// TIA Portal V17 export
// export: Created 2025-03-12T15:37:46.0301049Z, ExportSetting WithDefaults, DisplayName Totally Integrated Automation Portal, DisplayVersion V17 Update 8, DisplayName TIA Portal Openness, DisplayVersion V17 Update 8, DisplayName TIA Portal Version Control Interface, DisplayVersion V17, DisplayName SINAMICS Startdrive Advanced, DisplayVersion V17 SP2, DisplayName SINAMICS Startdrive G110M, G120, G120C, G120D, G120P, G115D, DisplayVersion V17 SP2, DisplayName SINAMICS Startdrive G130, G150, S120, S150, SINAMICS MV, S210, DisplayVersion V17 SP2, DisplayName STEP 7 Professional, DisplayVersion V17 Update 8, DisplayName SINUMERIK ONE STEP 7 Toolbox, DisplayVersion V17 Update 12, DisplayName SINUMERIK 840D sl STEP 7 Toolbox, DisplayVersion V17 Update 12, DisplayName STEP 7 Safety, DisplayVersion V17 Update 6, DisplayName WinCC Advanced, DisplayVersion V17 Update 8
TYPE "POWDER FEEDER HEATER JKT"
// stored: IsFailsafeCompliant false
   STRUCT
      START_GENERAL_CONDITIONS : Bool;   // Start General Conditions / START GENERAL CONDITIONS
      START_INITIAL_CONDITIONS_LINE_1 : Bool;   // Start Initial Conditions / START INITIAL CONDITIONS LINE 1
      START_INITIAL_CONDITIONS_LINE_2 : Bool;   // Start Initial Conditions / START INITIAL CONDITIONS LINE 2
      START_MANUAL_REQUEST_LINE_1 : Bool;   // Start Manual Request / START MANUAL REQUEST LINE 1
      START_MANUAL_REQUEST_LINE_2 : Bool;   // Start Manual Request / START MANUAL REQUEST LINE 2
      START_AUTO_REQUEST : Bool;   // Start Auto Request / START AUTO REQUEST
      START_GLOBAL_REQUEST_LINE_1 : Bool;   // Start Global Request / START GLOBAL REQUEST LINE 1
      START_GLOBAL_REQUEST_LINE_2 : Bool;   // Start Global Request / START GLOBAL REQUEST LINE 2
      START_COMMAND_LINE_1 : Bool;   // Start Command / START COMMAND LINE 1
      START_COMMAND_LINE_2 : Bool;   // Start Command / START COMMAND LINE 2
      START_LINE_1 : Bool;   // Start / START LINE 1
      START_LINE_2 : Bool;   // Start / START LINE 2
      FEEDBACK_ON_LINE_1 : Bool;   // Feedback On / FEEDBACK ON LINE 1
      FEEDBACK_ON_LINE_2 : Bool;   // Feedback On / FEEDBACK ON LINE 2
      STOP_GENERAL_CONDITIONS : Bool;   // Stop General Conditions / STOP GENERAL CONDITIONS
      STOP_INITIAL_CONDITIONS_LINE_1 : Bool;   // Stop Initial Conditions / STOP INITIAL CONDITIONS LINE 1
      STOP_INITIAL_CONDITIONS_LINE_2 : Bool;   // Stop Initial Conditions / STOP INITIAL CONDITIONS LINE 2
      STOP_MANUAL_REQUEST_LINE_1 : Bool;   // Stop Manual Request / STOP MANUAL REQUEST LINE 1
      STOP_MANUAL_REQUEST_LINE_2 : Bool;   // Stop Manual Request / STOP MANUAL REQUEST LINE 2
      STOP_AUTO_REQUEST : Bool;   // Stop Auto Request / STOP AUTO REQUEST
      STOP_GLOBAL_REQUEST_LINE_1 : Bool;   // Stop Global Request / STOP GLOBAL REQUEST LINE 1
      STOP_GLOBAL_REQUEST_LINE_2 : Bool;   // Stop Global Request / STOP GLOBAL REQUEST LINE 2
      STOP_COMMAND_LINE_1 : Bool;   // Stop Command / STOP COMMAND LINE 1
      STOP_COMMAND_LINE_2 : Bool;   // Stop Command / STOP COMMAND LINE 2
      STOP_LINE_1 : Bool;   // Stop / STOP LINE 1
      STOP_LINE_2 : Bool;   // Stop / STOP LINE 2
      FEEDBACK_OFF_LINE_1 : Bool;   // Feedback Off / FEEDBACK OFF LINE 1
      FEEDBACK_OFF_LINE_2 : Bool;   // Feedback Off / FEEDBACK OFF LINE 2
      START_GENERAL_CONDITIONS_HELP : Bool;   // Start General Conditions Help
      START_INITIAL_CONDITIONS_HELP : Bool;   // Start Initial Conditions Help
      STOP_GENERAL_CONDITIONS_HELP : Bool;   // Stop General Conditions Help
      STOP_INITIAL_CONDITIONS_HELP : Bool;   // Stop Initial Conditions Help
      FAULT : Bool;   // Fault
   END_STRUCT;
END_TYPE
